{attribute 'linkalways'} 
{attribute 'no_explicit_call' := 'This FB is a CLASS and must be accessed using methods or properties'}
{attribute 'enable_dynamic_creation'}
FUNCTION_BLOCK _Array0to1OfDINT EXTENDS ArrayDatatypeBase
VAR CONSTANT
	lBound : DINT := 0;
	uBound : DINT := 1;
END_VAR
VAR
	localData : ARRAY [lBound..uBound] OF DINT;
	activeData : REFERENCE TO ARRAY [lBound..uBound] OF DINT REF= localData;
	elements : ARRAY [lBound..uBound] OF _DINT(0);
	baseType : _DINT(0);
END_VAR

PROPERTY PUBLIC Address : PVOID
GET
Address := ADR(activeData);
END_GET
END_PROPERTY

PROPERTY PUBLIC BaseDatatype : I_Datatype
GET
BaseDatatype := baseType;
END_GET
END_PROPERTY

METHOD PUBLIC ClearReference
VAR_INPUT
END_VAR
activeData REF= localData;
SetElementReference();
END_METHOD

METHOD PUBLIC Clone : I_Datatype
VAR
    pClone : POINTER TO _Array0to1OfDINT;
END_VAR
pClone := __NEW(_Array0to1OfDINT());
pClone^.Value := Value;
Clone := pClone^;
END_METHOD

METHOD FB_init : BOOL
VAR_INPUT
	bInitRetains : BOOL; // if TRUE, the retain variables are initialized (warm start / cold start)
	bInCopyCode : BOOL;  // if TRUE, the instance afterwards gets moved into the copy code (online change)
END_VAR
SetElementReference();
END_METHOD

METHOD PUBLIC GetElementAsDatatypeByIndex : I_Datatype
VAR_INPUT
	Index : DINT;
END_VAR
GetElementAsDatatypeByIndex := elements[Index];
END_METHOD

METHOD PUBLIC GetElementByIndex : REFERENCE TO _DINT;
VAR_INPUT
	Index : DINT;
END_VAR
GetElementByIndex REF= elements[Index];
END_METHOD

PROPERTY PUBLIC LowerBound : DINT
GET
LowerBound := lBound;
END_GET
END_PROPERTY

METHOD PUBLIC MakeReferenceTo
VAR_INPUT
	ReferenceTarget : REFERENCE TO ARRAY [lBound..uBound] OF DINT;
END_VAR
activeData REF= ReferenceTarget;
SetElementReference();
END_METHOD

METHOD PROTECTED OnSerializeArrayValues
VAR_INPUT
	Serializer : I_Serializer;
END_VAR
VAR
	i : DINT;
END_VAR
FOR i := lBound TO uBound DO
	elements[i].SerializeWith(Serializer);
END_FOR
END_METHOD

METHOD PROTECTED SetElementReference
VAR_INPUT
END_VAR
VAR
	i : DINT;
END_VAR
FOR i := lBound TO uBound DO
	elements[i].MakeReferenceTo(activeData[i]);
END_FOR
END_METHOD

PROPERTY PUBLIC Size : UDINT
GET
Size := SIZEOF(activeData);
END_GET
END_PROPERTY

METHOD PROTECTED TryDeserializeArrayValues : BOOL
VAR_INPUT
	Deserializer : I_Deserializer;
	Feedback : I_DeserializerFeedback;
END_VAR
VAR
	enumerator : I_DeserializerArrayForwardEnumerator;
	i : DINT;
END_VAR
enumerator := Deserializer.GetArrayEnumerator();
i := lBound;

WHILE enumerator.MoveNext() AND i <= uBound DO
	
	IF NOT elements[i].TryDeserializeFrom(enumerator.Current, Feedback) THEN
		EXIT;
	END_IF
	i := i + 1;

END_WHILE
enumerator.Dispose();
END_METHOD

METHOD TryMakeReferenceTo : BOOL
VAR_INPUT
	Target : I_Datatype;
END_VAR
VAR
	targetAsArray : I_ArrayDatatype;
	pTargetData : POINTER TO ARRAY [lBound..uBound] OF DINT;
END_VAR
IF NOT Target.TryResolveAsArrayDatatype(targetAsArray) THEN
	RETURN;
END_IF

IF NOT (targetAsArray.Identifier = Identifier) THEN
	RETURN;
END_IF

pTargetData := Target.Address;
activeData REF= pTargetData^;
SetElementReference();
TryMakeReferenceTo := TRUE;
END_METHOD

PROPERTY PUBLIC UpperBound : DINT
GET
UpperBound := ubound;
END_GET
END_PROPERTY

PROPERTY PUBLIC Value : REFERENCE TO ARRAY [lBound..uBound] OF DINT;
GET
Value ref= activeData;
END_GET
END_PROPERTY

END_FUNCTION_BLOCK

(* stored: Version 1.1.0.1, ProductVersion 3.1.4024.13
   POU _Array0to1OfDINT: Id {04116934-13ab-050b-00a4-03ef308ac515}, SpecialFunc None
   Folder Core: Id {43c4ba50-f64a-0b8b-30fd-1a6d1807483b}
   Folder Constructor: Id {7410d06b-96a0-0459-184b-66f11a98fe5a}
   Folder Protected: Id {a84e7cf0-a8df-0577-3310-3e786475249e}
   Folder Customize: Id {88ba6ca0-79b6-0ac6-29e3-a1b90c09d5f4}
   Property Address: Id {3e492e45-7c2b-0402-0f3a-feb0d1540948}
   Get Get: Id {ea8dd621-9f2f-0f38-0005-d1bfb7624543}
   Property BaseDatatype: Id {a79cd5ff-d7fc-0d31-02d6-15adc9d30aef}
   Get Get: Id {02ec0351-06e7-0f1d-32a5-e4a014e3310e}
   Method ClearReference: Id {9ed911a9-c504-0bae-1790-e91634f1d8b7}
   Method Clone: Id {a692bc0a-278c-0046-0f76-ebd148cffd6a}
   Method FB_init: Id {492e93da-bd72-0295-0a3c-dc2cac461487}
   Method GetElementAsDatatypeByIndex: Id {0f7f8e08-40f3-09d7-31f9-ad987cb383c9}
   Method GetElementByIndex: Id {53323528-9cb7-0bde-00b5-4f60053ebb99}
   Property LowerBound: Id {37f51760-b2cd-0783-32cc-c68b828fab05}
   Get Get: Id {c600cee2-5016-0032-2d00-8b583e10ec40}
   Method MakeReferenceTo: Id {9e27c148-ad2b-0b65-2d7f-ab4071d38e42}
   Method OnSerializeArrayValues: Id {9de2c060-2bc2-0654-07d3-f657951831fe}
   Method SetElementReference: Id {3537e301-fdbf-4d27-bc3b-e5a57196ed77}
   Property Size: Id {3df9c90b-5975-05aa-15e0-8f2481c7480a}
   Get Get: Id {3fce2101-4062-0fe5-3305-2714342c2038}
   Method TryDeserializeArrayValues: Id {8df75494-f176-03ff-2304-d0f958db3cf5}
   Method TryMakeReferenceTo: Id {29e53d4d-535b-01ea-0307-6ce40a60fa38}
   Property UpperBound: Id {75ca5aaa-3645-06e8-31c9-ea5afd289856}
   Get Get: Id {9c048724-0caf-0800-1149-0fac7cdc5663}
   Property Value: Id {2ce8155d-7f66-06b6-3502-2baee3f8f8eb}
   Get Get: Id {761f0404-c759-05a2-2618-3c3cd8beb2d7} *)
